(* PLC project FbdBlockProject *)

PROGRAM FbdBlock
  VAR  (* added by the conversion: wires and edge detectors of the diagram *)
    _AND2_OUT : BOOL;
  END_VAR

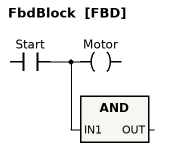
(* FBD diagram, written out as Structured Text *)
Motor := Start;
_AND2_OUT := AND(Start);
END_PROGRAM

CONFIGURATION Config
  RESOURCE Res ON PLC
  END_RESOURCE
END_CONFIGURATION
